TYPE "ValveCtrl"
VERSION : 0.1
// Block: ValveCtrl
   STRUCT
      SafeStop : Bool;
      Rst : Bool;
      MoveRest : Bool;
      MoveWork : Bool;
   END_STRUCT;

END_TYPE
